// SIMATIC S7-200 project (STEP 7-Micro/WIN), CPU 221 REL 01.10

SYMBOL_TABLE USER1
START            I0.0
MARK1            M0.0
MARK2            M0.1
GL1              Q0.0     // GreenLightL1
RL2              Q0.1     // RedLightL2
RL3              Q0.2     // RedLightL3
RL4              Q0.3     // RedLightL4
YL1              Q0.4     // YellowLightL1
YL2              Q0.5     // YellowLightL2
YL3              Q0.6     // YellowLightL3
YL4              Q0.7     // YellowLightL4
RL1              Q1.0     // RedLightL1
GL2              Q1.1     // GreenLightL2
GL3              Q1.2     // GreenLightL3
GL4              Q1.3     // GreenLightL4
END_SYMBOL_TABLE

ORGANIZATION_BLOCK MAIN:OB1
TITLE=PROGRAM COMMENTS
BEGIN
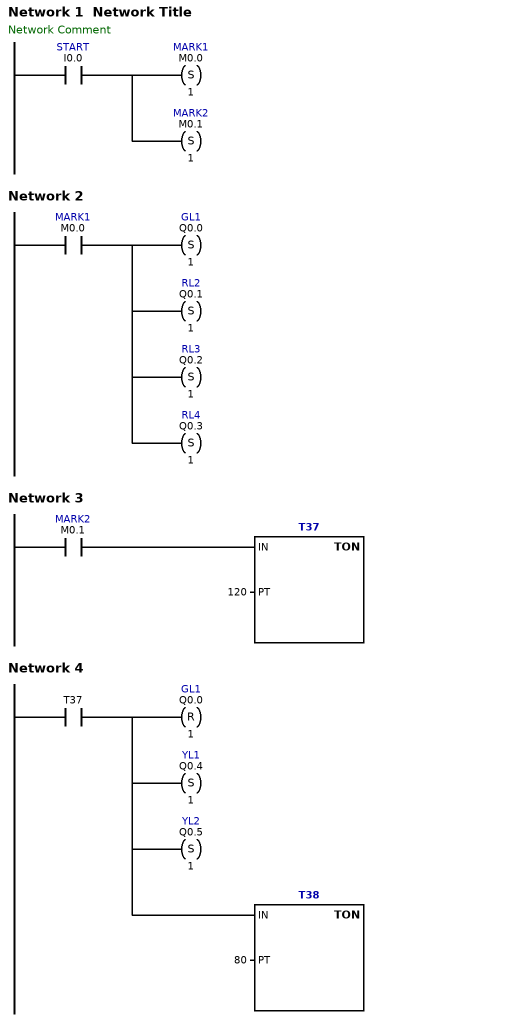
Network 1 // Network Title
// Network Comment
LD     START:I0.0
S      MARK1:M0.0, 1
S      MARK2:M0.1, 1
Network 2
LD     MARK1:M0.0
S      GL1:Q0.0, 1
S      RL2:Q0.1, 1
S      RL3:Q0.2, 1
S      RL4:Q0.3, 1
Network 3
LD     MARK2:M0.1
TON    T37, 120
Network 4
LD     T37
R      GL1:Q0.0, 1
S      YL1:Q0.4, 1
S      YL2:Q0.5, 1
TON    T38, 80
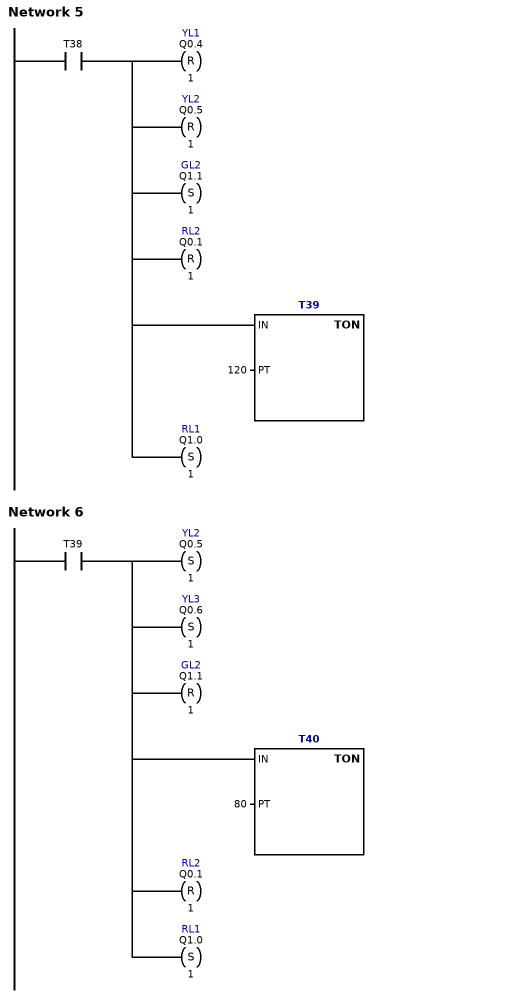
Network 5
LD     T38
R      YL1:Q0.4, 1
R      YL2:Q0.5, 1
S      GL2:Q1.1, 1
R      RL2:Q0.1, 1
TON    T39, 120
S      RL1:Q1.0, 1
Network 6
LD     T39
S      YL2:Q0.5, 1
S      YL3:Q0.6, 1
R      GL2:Q1.1, 1
TON    T40, 80
R      RL2:Q0.1, 1
S      RL1:Q1.0, 1
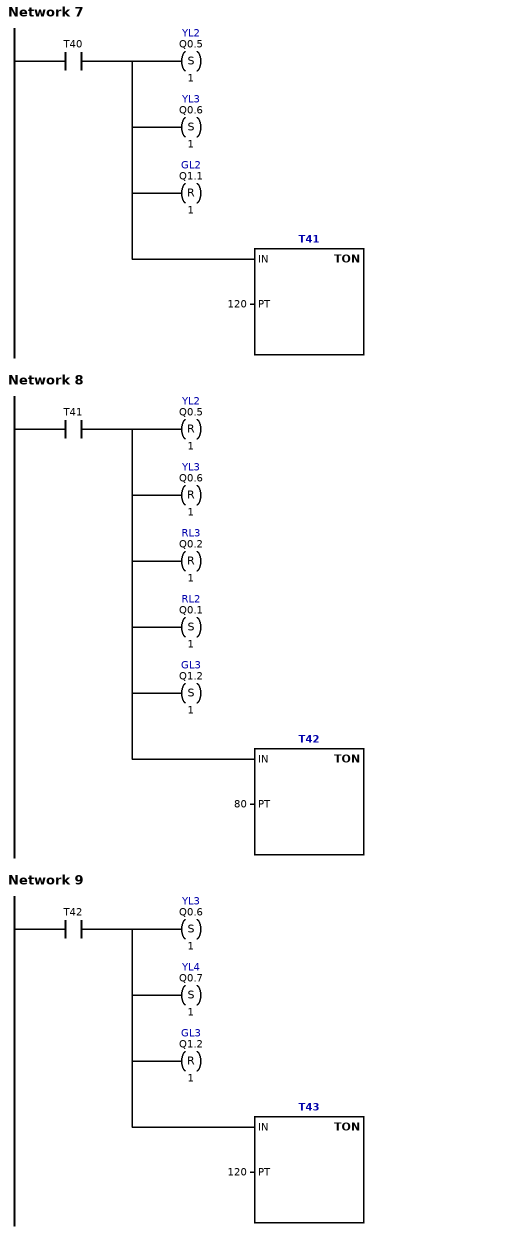
Network 7
LD     T40
S      YL2:Q0.5, 1
S      YL3:Q0.6, 1
R      GL2:Q1.1, 1
TON    T41, 120
Network 8
LD     T41
R      YL2:Q0.5, 1
R      YL3:Q0.6, 1
R      RL3:Q0.2, 1
S      RL2:Q0.1, 1
S      GL3:Q1.2, 1
TON    T42, 80
Network 9
LD     T42
S      YL3:Q0.6, 1
S      YL4:Q0.7, 1
R      GL3:Q1.2, 1
TON    T43, 120
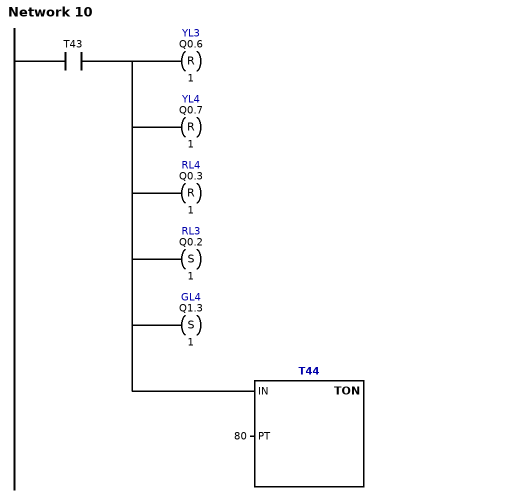
Network 10
LD     T43
R      YL3:Q0.6, 1
R      YL4:Q0.7, 1
R      RL4:Q0.3, 1
S      RL3:Q0.2, 1
S      GL4:Q1.3, 1
TON    T44, 80
END_ORGANIZATION_BLOCK
